TYPE FsT_PlcTaskInfo : FsST_PlcTaskInformation; END_TYPE

(* stored: Version 1.1.0.1, ProductVersion 3.1.4024.4
   DUT FsT_PlcTaskInfo: Id {b7f6a387-27a5-4c5a-860e-fee5f2e313e6} *)
